SUBAPPLICATION doppeltwirkend (* Subapplication Type *)
  (* Standard: 61499-2 *)
  (* Version 1.0, 2023-01-29, Franz *)
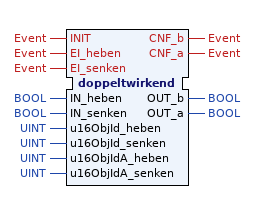
  EVENT_INPUT
    INIT;
    EI_heben;
    EI_senken;
  END_EVENT
  EVENT_OUTPUT
    CNF_b;
    CNF_a;
  END_EVENT
  VAR_INPUT
    IN_heben : BOOL;
    IN_senken : BOOL;
    u16ObjId_heben : UINT;
    u16ObjId_senken : UINT;
    u16ObjIdA_heben : UINT;
    u16ObjIdA_senken : UINT;
  END_VAR
  VAR_OUTPUT
    OUT_b : BOOL;
    OUT_a : BOOL;
  END_VAR
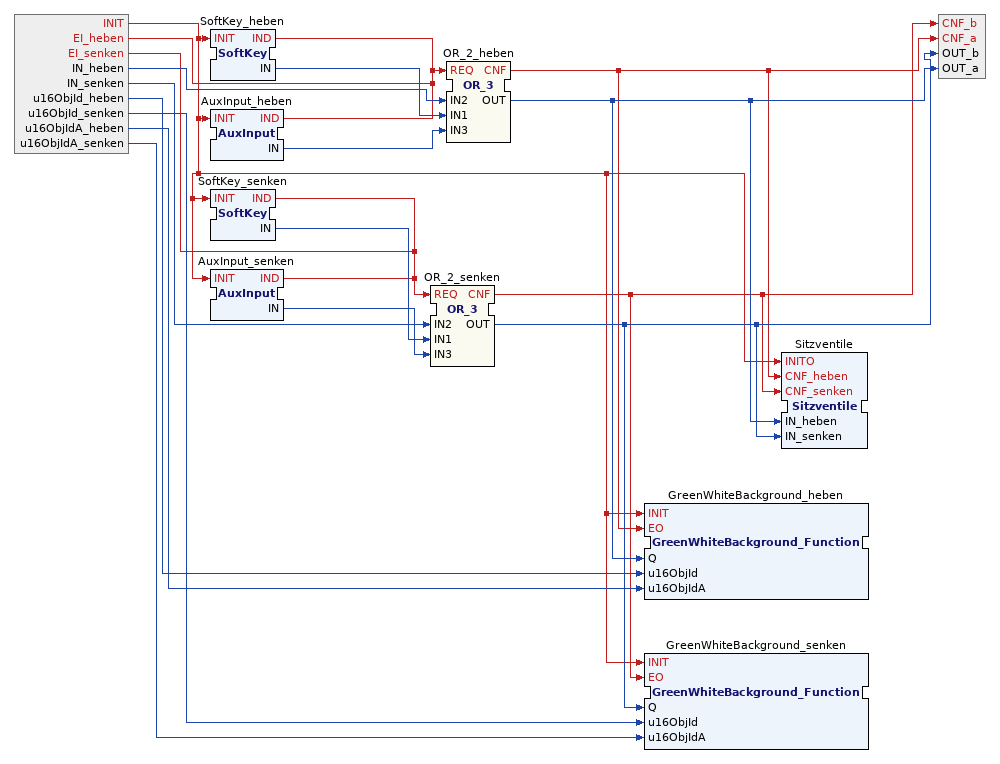
  FBS
    OR_2_heben : OR_3;
    OR_2_senken : OR_3;
  END_FBS
  SUBAPPS
    SoftKey_heben : SoftKey;
    SoftKey_senken : SoftKey;
    GreenWhiteBackground_heben : GreenWhiteBackground_Function;
    GreenWhiteBackground_senken : GreenWhiteBackground_Function;
    AuxInput_heben : AuxInput;
    AuxInput_senken : AuxInput;
    Sitzventile : Sitzventile;
  END_SUBAPPS
  EVENT_CONNECTIONS
    EI_heben TO OR_2_heben.REQ;
    OR_2_heben.CNF TO CNF_a;
    EI_senken TO OR_2_senken.REQ;
    OR_2_senken.CNF TO CNF_b;
    INIT TO SoftKey_heben.INIT;
    SoftKey_heben.IND TO OR_2_heben.REQ;
    INIT TO SoftKey_senken.INIT;
    SoftKey_senken.IND TO OR_2_senken.REQ;
    INIT TO GreenWhiteBackground_heben.INIT;
    OR_2_heben.CNF TO GreenWhiteBackground_heben.EO;
    INIT TO GreenWhiteBackground_senken.INIT;
    OR_2_senken.CNF TO GreenWhiteBackground_senken.EO;
    INIT TO AuxInput_heben.INIT;
    AuxInput_heben.IND TO OR_2_heben.REQ;
    INIT TO AuxInput_senken.INIT;
    AuxInput_senken.IND TO OR_2_senken.REQ;
    INIT TO Sitzventile.INITO;
    OR_2_heben.CNF TO Sitzventile.CNF_heben;
    OR_2_senken.CNF TO Sitzventile.CNF_senken;
  END_CONNECTIONS
  DATA_CONNECTIONS
    IN_heben TO OR_2_heben.IN2;
    OR_2_heben.OUT TO OUT_a;
    IN_senken TO OR_2_senken.IN2;
    OR_2_senken.OUT TO OUT_b;
    SoftKey_heben.IN TO OR_2_heben.IN1;
    SoftKey_senken.IN TO OR_2_senken.IN1;
    OR_2_heben.OUT TO GreenWhiteBackground_heben.Q;
    OR_2_senken.OUT TO GreenWhiteBackground_senken.Q;
    u16ObjId_heben TO GreenWhiteBackground_heben.u16ObjId;
    u16ObjId_senken TO GreenWhiteBackground_senken.u16ObjId;
    u16ObjIdA_heben TO GreenWhiteBackground_heben.u16ObjIdA;
    u16ObjIdA_senken TO GreenWhiteBackground_senken.u16ObjIdA;
    AuxInput_heben.IN TO OR_2_heben.IN3;
    AuxInput_senken.IN TO OR_2_senken.IN3;
    OR_2_heben.OUT TO Sitzventile.IN_heben;
    OR_2_senken.OUT TO Sitzventile.IN_senken;
  END_CONNECTIONS
END_SUBAPPLICATION
